// Returns the name of a variable as a string using its pointer and size.
// Variables allocated in dynamic memory are not supported.
FUNCTION FsF_GetVariablePath : FsT_Str
VAR_INPUT
	Variable : ANY;
END_VAR
VAR
	nTmp : UDINT := SIZEOF(FsF_GetVariablePath);
END_VAR

_FsGVL.fbTcComIecApplicationInfo
	.GetInterface()
	.GetSymbolNameByAddress(TO_UDINT(Variable.diSize), Variable.pValue, nTmp, ADR(FsF_GetVariablePath));

END_FUNCTION

(* stored: Version 1.1.0.1, ProductVersion 3.1.4024.4
   POU FsF_GetVariablePath: Id {48e3408e-4798-4cb5-abb4-4adc1df265d4}, SpecialFunc None *)
